DATA_BLOCK "ton_timer_t"
{InstructionName := 'IEC_TIMER';
LibVersion := '1.0';
S7_Optimized_Access := 'true' }
AUTHOR : Simatic
FAMILY : IEC
NAME : IEC_TMR
VERSION : 1.0
NON_RETAIN
IEC_TIMER

BEGIN

END_DATA_BLOCK

